TYPE AlarmLog :
STRUCT
	Head: INT;
	Tail: INT;
	Alarms: ARRAY [Globals.AlarmsLow..Globals.AlarmsHigh] OF AlarmEvent;
END_STRUCT
END_TYPE

(* stored: Version 1.1.0.1, ProductVersion 3.1.4024.5
   DUT AlarmLog: Id {d54d625d-5743-43c4-a890-62c7cb5e28f1} *)
